PROGRAM PRG_Compilation
VAR

	
END_VAR

END_PROGRAM

(* stored: Version 1.1.0.1
   POU PRG_Compilation: Id {5db94455-dadb-0232-2011-e8c0ba8c59a8}, SpecialFunc None *)
